PROGRAM JIG_EMPTY
VAR
END_VAR

END_PROGRAM

(* stored: Version 1.1.0.1, ProductVersion 3.1.4022.18
   POU JIG_EMPTY: Id {8a99bef7-1401-4a01-b48b-622eed1dfbdc}, SpecialFunc None *)
